FUNCTION_BLOCK FB_DrukknopSpecial
VAR_INPUT
    bDrukknop : BOOL;          // fysiek knopsignaal
END_VAR

VAR_OUTPUT
    bSingle    : BOOL;
    bDouble    : BOOL;
    bLong      : BOOL;
END_VAR

VAR
    fbSD : FB_SingleDoubleClick;
    fbSL : FB_ShortLongClick;
END_VAR

// --- Doorgeven van de knop als input ---
fbSD(bSwitch := bDrukknop, tSwitchTime := T#500MS);
fbSL(bSwitch := bDrukknop, tSwitchTime := T#1S);

// --- Outputs ---
bSingle := fbSD.bSingleClick AND NOT fbSL.bLongClick;
bDouble := fbSD.bDoubleClick;
bLong   := fbSL.bLongClick;

END_FUNCTION_BLOCK

(* stored: Version 1.1.0.1, ProductVersion 3.1.4024.15
   POU FB_DrukknopSpecial: Id {e3bfc8b3-48b0-41ec-970b-bff868bbde04}, SpecialFunc None *)
